// TIA Portal project "Format_Time" (V18)

(* hardware
DEVICE "S7-1200 station_1"  S7-1200 Station
   slot 0: "Rack_0"  S7-1200 Rack  Rack  V1.0
   slot 1: "PLC_1"  CPU 1214C DC/DC/DC  6ES7 214-1AG40-0XB0  V4.5
DEVICE "HMI_1"  KTP700 Basic PN
   slot 0: "HMI_1"  KTP700 Basic PN  6AV2 123-2GB03-0AX0  17.0.0.0
   slot 1: "HMI_RT_1"  KTP700 Basic PN  6AV2 123-2GB03-0AX0  17.0.0.0
   slot 5: "HMI_1.IE_CP_1"  PROFINET Interface  17.0.0.0
      slot 1: "PROFINET Interface_1"  PROFINET Interface
         slot 1: "Port_1"  Port
*)

// ===== PLC "PLC_1"  CPU 1214C DC/DC/DC =====

VAR_GLOBAL   // PLC tag table "Default tag table"
   "System_Byte" AT %MB1 : Byte;
   "FirstScan" AT %M1.0 : Bool;
   "DiagStatusUpdate" AT %M1.1 : Bool;
   "AlwaysTRUE" AT %M1.2 : Bool;
   "AlwaysFALSE" AT %M1.3 : Bool;
   "Clock_Byte" AT %MB0 : Byte;
   "Clock_10Hz" AT %M0.0 : Bool;
   "Clock_5Hz" AT %M0.1 : Bool;
   "Clock_2.5Hz" AT %M0.2 : Bool;
   "Clock_2Hz" AT %M0.3 : Bool;
   "Clock_1.25Hz" AT %M0.4 : Bool;
   "Clock_1Hz" AT %M0.5 : Bool;
   "Clock_0.625Hz" AT %M0.6 : Bool;
   "Clock_0.5Hz" AT %M0.7 : Bool;
END_VAR

// folder: DBs

DATA_BLOCK "Var_IHM"   // DB1
{ S7_Optimized_Access := 'TRUE' }
VERSION : 0.1
   VAR
      Tela_Root : Struct
         Bt_Liga_Timer1 : Bool;
         Bt_Liga_Timer2 : Bool;
         Current_Timer1 : Time;
         Current_Timer2 : Time;
         Secounds_Timer1 : Int;
         Minutes_Timer1 : Int;
         Hours_Timer1 : Int;
         Secounds_Timer2 : Int;
         Minutes_Timer2 : Int;
         Hours_Timer2 : Int;
      END_STRUCT;
   END_VAR
BEGIN
END_DATA_BLOCK

// folder: System blocks/Program resources

DATA_BLOCK "IEC_Timer_1_DB"   // DB2
{ S7_Optimized_Access := 'TRUE' }
AUTHOR : Simatic
FAMILY : IEC
NAME : IEC_TMR
VERSION : 1.0
// stored: InstanceOfName IEC_TIMER
"IEC_TIMER"
BEGIN
END_DATA_BLOCK

DATA_BLOCK "IEC_Timer_2_DB"   // DB3
{ S7_Optimized_Access := 'TRUE' }
AUTHOR : Simatic
FAMILY : IEC
NAME : IEC_TMR
VERSION : 1.0
// stored: InstanceOfName IEC_TIMER
"IEC_TIMER"
BEGIN
END_DATA_BLOCK

// folder: (top level)

ORGANIZATION_BLOCK "Main"   // OB1, LAD, ProgramCycle
TITLE = "Main Program Sweep (Cycle)"
{ S7_Optimized_Access := 'TRUE' }
VERSION : 0.1
   VAR_INPUT
      Initial_Call : Bool;   // Initial call of this OB
      Remanence : Bool;   // =True, if remanent data are available
   END_VAR
   VAR_TEMP   // added for the SCL form of the ladder/FBD networks
      _w1 : Bool;
   END_VAR
BEGIN

REGION Network 1
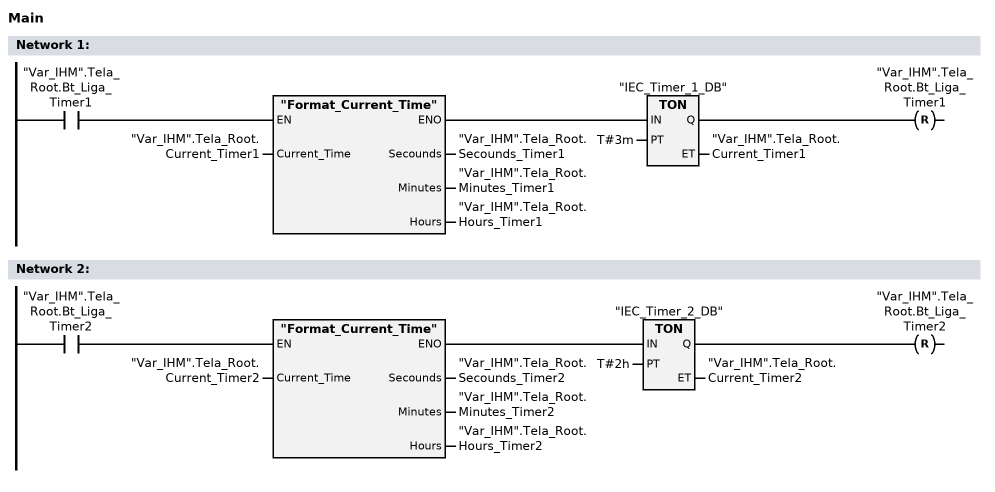
   "Format_Current_Time"(EN := "Var_IHM".Tela_Root.Bt_Liga_Timer1,
                         Current_Time := "Var_IHM".Tela_Root.Current_Timer1,
                         Secounds => "Var_IHM".Tela_Root.Secounds_Timer1,
                         Minutes => "Var_IHM".Tela_Root.Minutes_Timer1,
                         Hours => "Var_IHM".Tela_Root.Hours_Timer1,
                         ENO => #_w1);
   "IEC_Timer_1_DB".TON(IN := #_w1, PT := T#3m, ET => "Var_IHM".Tela_Root.Current_Timer1);
   IF "IEC_Timer_1_DB".Q THEN "Var_IHM".Tela_Root.Bt_Liga_Timer1 := FALSE; END_IF;
END_REGION

REGION Network 2
   "Format_Current_Time"(EN := "Var_IHM".Tela_Root.Bt_Liga_Timer2,
                         Current_Time := "Var_IHM".Tela_Root.Current_Timer2,
                         Secounds => "Var_IHM".Tela_Root.Secounds_Timer2,
                         Minutes => "Var_IHM".Tela_Root.Minutes_Timer2,
                         Hours => "Var_IHM".Tela_Root.Hours_Timer2,
                         ENO => #_w1);
   "IEC_Timer_2_DB".TON(IN := #_w1, PT := T#2h, ET => "Var_IHM".Tela_Root.Current_Timer2);
   IF "IEC_Timer_2_DB".Q THEN "Var_IHM".Tela_Root.Bt_Liga_Timer2 := FALSE; END_IF;
END_REGION
END_ORGANIZATION_BLOCK

// folder: FCs

FUNCTION "Format_Current_Time" : Void   // FC1, SCL
{ S7_Optimized_Access := 'TRUE' }
AUTHOR : Ezequiel
VERSION : 0.1
   VAR_INPUT
      Current_Time : Time;
   END_VAR
   VAR_OUTPUT
      Secounds : Int;
      Minutes : Int;
      Hours : Int;
   END_VAR
   VAR_TEMP
      Total_Segundos : Int;
      Tempo_DINT : DInt;
      Total_Segundos_Real : Real;
   END_VAR
BEGIN
   #Tempo_DINT := TIME_TO_DINT(#Current_Time);
   #Total_Segundos_Real := #Tempo_DINT / 1000;
   #Secounds := (#Tempo_DINT / 1000) MOD 60;
   #Minutes := ((#Tempo_DINT / 1000) / 60) MOD 60;
   #Hours := DINT_TO_INT(TRUNC(#Total_Segundos_Real / 3600));
END_FUNCTION

(* ===== HMI "HMI_RT_1" =====
system functions are stored by id; their names below are inferred from use
connection "HMI_Connection_1": ETHERNET, SMART_S7_1200_OMS

HMI tags "Default tag table"
   "Tag_ScreenNumber" : UInt, internal
   "Var_IHM_Tela_Root_Bt_Liga_Timer1" : Bool = PLC Var_IHM.Tela_Root.Bt_Liga_Timer1, 1 s
   "Var_IHM_Tela_Root_Bt_Liga_Timer2" : Bool = PLC Var_IHM.Tela_Root.Bt_Liga_Timer2, 1 s
   "Var_IHM_Tela_Root_Current_Timer1" : Time = PLC Var_IHM.Tela_Root.Current_Timer1, 1 s
   "Var_IHM_Tela_Root_Hours_Timer1" : Int = PLC Var_IHM.Tela_Root.Hours_Timer1, 1 s
   "Var_IHM_Tela_Root_Minutes_Timer1" : Int = PLC Var_IHM.Tela_Root.Minutes_Timer1, 1 s
   "Var_IHM_Tela_Root_Secounds_Timer1" : Int = PLC Var_IHM.Tela_Root.Secounds_Timer1, 1 s
   "Var_IHM_Tela_Root_Secounds_Timer2" : Int = PLC Var_IHM.Tela_Root.Secounds_Timer2, 1 s
   "Var_IHM_Tela_Root_Hours_Timer2" : Int = PLC Var_IHM.Tela_Root.Hours_Timer2, 1 s
   "Var_IHM_Tela_Root_Minutes_Timer2" : Int = PLC Var_IHM.Tela_Root.Minutes_Timer2, 1 s

Template "Template_1" 800x480
   Button "Alarms" at 714,429 size 71x50; TextOff 'Alarms'; PictureOff "AlarmDisplay_KTP700_Basic_PN_TR"; PictureOn "AlarmDisplay_KTP700_Basic_PN_TR"
      on Release: function_ef3f5d25("Alarm window_Unacknowledged", -1)
   Button "Template_Button" at 614,429 size 71x50; TextOff 'Text'
   Button "Template_Button_1" at 514,429 size 71x50; TextOff 'Text'
   Button "Template_Button_2" at 414,429 size 71x50; TextOff 'Text'
   Button "Template_Button_3" at 314,429 size 71x50; TextOff 'Text'
   Button "Template_Button_4" at 214,429 size 71x50; TextOff 'Text'
   Button "Template_Button_5" at 114,429 size 71x50; TextOff 'Text'
   Button "Start screen" at 14,429 size 71x50; TextOff 'Start screen'; PictureOff "NavigateHome_KTP700_Basic_PN_TR"; PictureOn "NavigateHome_KTP700_Basic_PN_TR"
      on Release: ActivateScreen("Root screen", 0)
   SymbolicIOField "Symbolic_IO_Field_Screen" at 93,9 size 600x33; TextOff '0'; TextOn '1'; TextList "TextList_ScreenNames"
      ProcessValue <- "Tag_ScreenNumber"
      on Change: ActivateScreenByNumber("Tag_ScreenNumber", 0)
   DateTimeField "HmiScreenItemData" at 695,25 size 105x25
   DateTimeField "HmiScreenItemData_1" at 695,0 size 105x25
   GraphicView "Logo" at 0,0 size 91x51; Picture "Logo of HMI_1"

screen "Root screen" 800x480, template "Template_1"
   on GenerateScreen: SetTag("Tag_ScreenNumber", 1)
   Button "HmiScreenItemData_1" at 17,49 size 159x47; TextOff 'System screens'; PictureOff "Navigates to System screens for KTP700 Basic+ PN 17.0.0.0"; PictureOn "Navigates to System screens for KTP700 Basic+ PN 17.0.0.0"
      on Release: ActivateScreen("System screens", 0)
   Switch "Switch_1" at 226,240 size 103x32; CaptionText 'Switch'; TextOff 'OFF'; TextOn 'ON'
      ProcessValue <- "Var_IHM_Tela_Root_Bt_Liga_Timer1"
   Switch "Switch_2" at 519,240 size 102x32; CaptionText 'Switch'; TextOff 'OFF'; TextOn 'ON'
      ProcessValue <- "Var_IHM_Tela_Root_Bt_Liga_Timer2"
   TextField "Text field_1" at 246,206 size 68x23; Text 'Timer 1'
   TextField "Text field_2" at 536,206 size 68x23; Text 'Timer 2'
   IOField "I/O field_1" at 232,304 size 32x37; FormatPattern 99; Unit :
      ProcessValue <- "Var_IHM_Tela_Root_Hours_Timer1"
   IOField "I/O field_2" at 260,304 size 32x37; FormatPattern 99; Unit :
      ProcessValue <- "Var_IHM_Tela_Root_Minutes_Timer1"
   IOField "I/O field_3" at 288,304 size 32x37; FormatPattern 99
      ProcessValue <- "Var_IHM_Tela_Root_Secounds_Timer1"
   IOField "I/O field_4" at 524,304 size 32x37; FormatPattern 99; Unit :
      ProcessValue <- "Var_IHM_Tela_Root_Hours_Timer2"
   IOField "I/O field_5" at 552,304 size 32x37; FormatPattern 99; Unit :
      ProcessValue <- "Var_IHM_Tela_Root_Minutes_Timer2"
   IOField "I/O field_6" at 580,304 size 32x37; FormatPattern 99
      ProcessValue <- "Var_IHM_Tela_Root_Secounds_Timer2"

screen "System screens" 800x480, template "Template_1"
   on GenerateScreen: SetTag("Tag_ScreenNumber", 2)
   Button "Back" at 1,52 size 159x47; TextOff 'Back'
      on Release: ActivateScreen("Root screen", 0)
   Button "HmiScreenItemData" at 36,146 size 159x47; TextOff 'SIMATIC PLC system diagnos...'; PictureOff "Navigates to SIMATIC PLC system diagnostics for KTP700 Basic+ PN 17.0.0.0"; PictureOn "Navigates to SIMATIC PLC system diagnostics for KTP700 Basic+ PN 17.0.0.0"
      on Release: ActivateScreen("SIMATIC PLC system diagnostics", 0)
   Button "HmiScreenItemData_1" at 36,205 size 159x47; TextOff 'Project information'; PictureOff "Navigates to Project information for KTP700 Basic+ PN 17.0.0.0"; PictureOn "Navigates to Project information for KTP700 Basic+ PN 17.0.0.0"
      on Release: ActivateScreen("Project information", 0)
   Button "HmiScreenItemData_2" at 36,264 size 159x47; TextOff 'User administration'; PictureOff "Navigates to User administration for KTP700 Basic+ PN 17.0.0.0"; PictureOn "Navigates to User administration for KTP700 Basic+ PN 17.0.0.0"
      on Release: ActivateScreen("User administration", 0)
   Button "HmiScreenItemData_3" at 36,323 size 159x47; TextOff 'System information'; PictureOff "Navigates to System information for KTP700 Basic+ PN 17.0.0.0"; PictureOn "Navigates to System information for KTP700 Basic+ PN 17.0.0.0"
      on Release: ActivateScreen("System information", 0)

screen "SIMATIC PLC system diagnostics" 800x480, template "Template_1"
   on GenerateScreen: SetTag("Tag_ScreenNumber", 3)
   SysDiagControl "HmiScreenItemData" at 1,100 size 796x321
   Button "Back" at 1,52 size 159x47; TextOff 'Back'
      on Release: ActivateScreen("System screens", 0)

screen "Project information" 800x480, template "Template_1"
   on GenerateScreen: SetTag("Tag_ScreenNumber", 4)
   TextField "HmiScreenItemData" at 35,102 size 171x28; Text 'Project name:'
   TextField "HmiScreenItemData_1" at 241,102 size 524x28; Text 'Format_Time'
   TextField "HmiScreenItemData_2" at 35,132 size 171x28; Text 'Created on:'
   TextField "HmiScreenItemData_3" at 241,132 size 524x28; Text '8/29/2024 8:20:00 AM'
   TextField "HmiScreenItemData_4" at 35,162 size 171x28; Text 'Author:'
   TextField "HmiScreenItemData_5" at 241,162 size 524x28; Text 'Ezequiel'
   TextField "HmiScreenItemData_6" at 35,192 size 171x28; Text 'Description:'
   TextField "HmiScreenItemData_7" at 241,192 size 524x28; Text '(not configured)'
   Button "Back" at 1,52 size 159x47; TextOff 'Back'
      on Release: ActivateScreen("System screens", 0)

screen "User administration" 800x480, template "Template_1"
   on GenerateScreen: SetTag("Tag_ScreenNumber", 5)
   UserView "HmiScreenItemData" at 1,100 size 796x321
   Button "Back" at 1,52 size 159x47; TextOff 'Back'
      on Release: ActivateScreen("System screens", 0)

screen "System information" 800x480, template "Template_1"
   on GenerateScreen: SetTag("Tag_ScreenNumber", 6)
   TextField "HmiScreenItemData" at 35,102 size 171x28; Text 'HMI device type:'
   TextField "HmiScreenItemData_1" at 241,102 size 524x28; Text 'KTP700 Basic+ PN 17.0.0.0'
   TextField "HmiScreenItemData_2" at 35,132 size 171x28; Text 'Connection:'
   TextField "HmiScreenItemData_3" at 241,132 size 524x28; Text 'PROFINET (X1)'
   TextField "HmiScreenItemData_4" at 35,162 size 171x28; Text 'PLC:'
   TextField "HmiScreenItemData_5" at 241,162 size 524x28; Text 'SIMATIC S7 1200'
   Button "Back" at 1,52 size 159x47; TextOff 'Back'
      on Release: ActivateScreen("System screens", 0)
*)